FUNCTION_BLOCK FB_Unwind EXTENDS FB_PackML_BaseModule
VAR
	Axis	  : FB_Component_BasicSlaveAxis := (Name := 'Unwind Axis');
	MasterRef : REFERENCE TO AXIS_REF;
END_VAR

METHOD PROTECTED Aborting
// Mode is ignored
CASE SequenceState OF
	0:
		NoStateTasksToComplete := FALSE;
		SequenceState		   := SequenceState + 10;

	10: // Stop Axis
		Axis.Override := 100;
		Axis.Stop(); // This will also GearOut
		IF Axis.Stopped THEN
			SequenceState := SequenceState + 10;
		END_IF

	20: // Disable Axis
		Axis.Disable();
		IF NOT Axis.Enabled THEN
			SequenceState := SequenceState + 10;
		END_IF

	30:
		StateTasksComplete := TRUE;
END_CASE

SUPER^.Aborting();
END_METHOD

PROPERTY AxisRef : REFERENCE TO AXIS_REF
GET
AxisRef REF= Axis.Axis;
END_GET
END_PROPERTY

METHOD PROTECTED Completing
CASE _CurrentMode OF
	ePMLUnitMode_Production:
		CASE SequenceState OF
			0:
				NoStateTasksToComplete := FALSE;
				SequenceState		   := SequenceState + 10;

			10: // Wait for Master Axis to Stop and GearOut, or Stop
				IF Axis.InGear AND Axis.Stopped THEN
					Axis.GearOut();
				ELSIF NOT Axis.InGear THEN
					Axis.Stop();
				END_IF

				IF Axis.Stopped THEN
					SequenceState := SequenceState + 10;
				END_IF

			20:
				StateTasksComplete := TRUE;
		END_CASE

	ePMLProtUnitMode_Maintenance, ePMLProtUnitMode_Manual:
		;
END_CASE

SUPER^.Completing();
END_METHOD

METHOD PUBLIC CyclicLogic
IF NOT InitComplete THEN
	_InitComplete := Initialize();
	RETURN;
END_IF

SUPER^.CyclicLogic();
END_METHOD

METHOD PROTECTED Initialize : BOOL;
VAR
	i : UDINT;
END_VAR
Initialize := FALSE;
CASE DescendantSequenceState OF
	0: // Register Components
		RegisterComponent(Axis);

		// Set Config
		_LogModeChanges			:= FALSE;
		_LogStateChanges		:= FALSE;
		DescendantSequenceState := DescendantSequenceState + 10;

	10:
		// Copy Mode names
		FOR i := 1 TO 10 DO
			ModeNames[i] := F_UnitModeToString(UDINT_TO_INT(i));
		END_FOR

		DescendantSequenceState := DescendantSequenceState + 10;

	20:
		IF SUPER^.Initialize() THEN
			DescendantSequenceState := DescendantSequenceState + 10;
		END_IF

	30:
		Initialize := TRUE;
END_CASE
END_METHOD

PROPERTY MasterAxisRef : REFERENCE TO AXIS_REF
SET
MasterRef REF= MasterAxisRef;
END_SET
END_PROPERTY

METHOD PROTECTED Starting
CASE _CommandedMode OF
	ePMLProtUnitMode_Production:
		CASE SequenceState OF
			0:
				NoStateTasksToComplete := FALSE;
				SequenceState		   := SequenceState + 10;

			10: // Enable Axis
				Axis.Enable();
				IF Axis.Enabled THEN
					SequenceState := SequenceState + 10;
				END_IF

			20: // Set reference to Master and Couple Axes
				Axis.Master1	  REF= MasterRef;
				Axis.RatioMaster1 := 0.5; // Can be set at anytime and changed while in motion
				Axis.GearIn();
				IF Axis.InGear THEN
					SequenceState := SequenceState + 10;
				END_IF

			30:
				StateTasksComplete := TRUE;
		END_CASE
END_CASE

SUPER^.Starting();
END_METHOD

METHOD PROTECTED Stopping
CASE _CurrentMode OF
	ePMLUnitMode_Production:
		CASE SequenceState OF
			0:
				NoStateTasksToComplete := FALSE;
				SequenceState		   := SequenceState + 10;

			10: // Stop Axis
				Axis.Override := 100;
				Axis.Stop(); // This will also GearOut
				IF Axis.Stopped THEN
					SequenceState := SequenceState + 10;
				END_IF

			20:
				StateTasksComplete := TRUE;
		END_CASE
END_CASE

SUPER^.Stopping();
END_METHOD

END_FUNCTION_BLOCK

(* stored: Version 1.1.0.1, ProductVersion 3.1.4024.12
   POU FB_Unwind: Id {531fe024-1c35-49f6-9ea6-b83468bb853c}, SpecialFunc None
   Method Aborting: Id {0e94a613-0e2d-43e0-9b59-861775c0ebdb}
   Property AxisRef: Id {d13e3860-08f0-4ce9-b897-f8cfcdba7e93}
   Get Get: Id {e4cb4012-07fb-4a4b-a3d7-60c1cc05d1d7}
   Method Completing: Id {2b5befec-31ac-4e0e-8a6d-577805b741ec}
   Method CyclicLogic: Id {761193c7-ca9e-4580-b131-82e57b210c90}
   Method Initialize: Id {e3a8ca4b-f177-4610-88fe-7274fe30d43b}
   Property MasterAxisRef: Id {3374daa1-7f61-440f-abd3-569198fd16f3}
   Set Set: Id {5f9e248d-d1a0-4f8f-bf65-7d19780c479a}
   Method Starting: Id {edea4660-a85a-4b0f-83e4-8557ebe4b1fc}
   Method Stopping: Id {c55df479-e1d7-47c1-8f42-c67178fb7cf3} *)
